(* CODESYS project doser.project

Project tree, tasks and I/O mapping:
  Device : CODESYS Control Win V3, 3S - Smart Software Solutions GmbH, order no. 305021, version 3.5.5.50
    application Application
      libraries: Standard, * (System)
      task MainTask (cyclic, interval t#20ms, priority 1) calls GateTest
      program PLC_PRG [ST]
      Global_variables/
        global variables GL_AI
        global variables GL_AO
        global variables GL_DI
        global variables GL_DO
      Units/
        function block AnalogHandler [ST]
        function block MotorDriver [ST]
        function block ProductHandler [ST]
        function block ProximitySensor [ST]
        function block GateDriver [ST]
      Tests/
        program Motor_test [LD]
        program Proximity_test [LD]
        program GateTest [LD]
*)

// Device/Application/Global_variables/GL_AI
VAR_GLOBAL
	load_cell_1_ai :INT;
	load_cell_2_ai :INT;
	
END_VAR

// Device/Application/Global_variables/GL_AO
VAR_GLOBAL
	doser_motor_freq_1_ao :INT;
	doser_motor_freq_2_ao :INT;
	mixer_motor_freq_ao :INT;
END_VAR

// Device/Application/Global_variables/GL_DI
VAR_GLOBAL
	doser_motor_overload_1 :BOOL;
	doser_motor_overload_2 :BOOL;
	mixer_motor_overload_1 :BOOL;
	gate_is_open :BOOL;
	emgc :BOOL;
	
END_VAR

// Device/Application/Global_variables/GL_DO
VAR_GLOBAL
	do_doser_moter_coil_1:BOOL;
	do_doser_moter_coil_3:BOOL;
	do_mixer_moter_coil :BOOL;
	do_gate_coil:BOOL;	
END_VAR

// Device/Application/Tests/GateTest
PROGRAM GateTest
VAR
	GateDriver_0: GateDriver;
	act: BOOL;
	egv: BOOL;
	open: BOOL;
	time_open: TIME;
	timeout: TIME;
	fault: BOOL;
	state_open: BOOL;
END_VAR

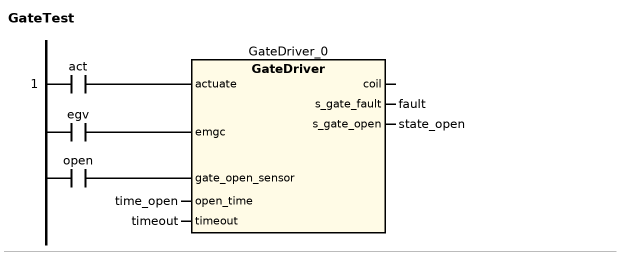
// NETWORK 1
GateDriver_0(
    actuate := act,
    emgc := egv,
    gate_open_sensor := open,
    open_time := time_open,
    timeout := timeout,
    s_gate_fault => fault,
    s_gate_open => state_open); // GateDriver

END_PROGRAM

// Device/Application/Units/GateDriver
FUNCTION_BLOCK GateDriver

VAR_INPUT
	actuate:BOOL;
	emgc:BOOL;
	gate_open_sensor:BOOL;
	open_time:TIME;
	timeout:TIME;
END_VAR


VAR_OUTPUT
	coil:BOOL;
	s_gate_fault:BOOL;
	s_gate_open:BOOL;
END_VAR


VAR
	gate_open_timeout:ton;
	gate_open_timer:ton;
	gate_trigger:r_trig;
	state:int;
END_VAR

CASE state OF
	0:
		coil:=FALSE;
		s_gate_fault:=FALSE;
		s_gate_open:=FALSE;
		gate_open_timeout(in:=FALSE);
		gate_open_timer(in:=FALSE);
		gate_trigger(clk:=actuate);
		IF gate_trigger.Q THEN
			state:=1;
			coil:=TRUE;
		END_IF
	
	1:
		gate_open_timeout(in:=TRUE, pt:=timeout);
		IF gate_open_sensor THEN
			s_gate_open:=TRUE;
			state:=2;
		ELSIF gate_open_timeout.Q THEN
			s_gate_fault:=TRUE;
			coil:=FALSE;
		END_IF
	
	2:
		gate_open_timer(in:=TRUE, pt:=open_time);
		IF gate_open_timer.Q THEN
			coil:=FALSE;
			s_gate_open:=FALSE;
		END_IF
END_CASE


IF emgc OR actuate=FALSE THEN
	state:=0;
END_IF

END_FUNCTION_BLOCK

// Device/Application/PLC_PRG
PROGRAM PLC_PRG
VAR
END_VAR

END_PROGRAM

// Device/Application/Units/AnalogHandler
FUNCTION_BLOCK AnalogHandler
VAR_INPUT
	AnalogSignal:INT;
	Gain:REAL;
	UpperLimit:REAL;
	LowerLimit:REAL;
	
END_VAR
VAR_OUTPUT
	ScaledValue:REAL;
	UpperLimitWarning:BOOL;
	LowerLimitWarning:BOOL;
END_VAR
VAR
END_VAR

ScaledValue := AnalogSignal * Gain;

IF ScaledValue > UpperLimit THEN
	UpperLimitWarning := TRUE;
ELSE
	UpperLimitWarning := FALSE;
END_IF


IF ScaledValue < LowerLimit THEN
	LowerLimitWarning := TRUE;
ELSE
	LowerLimitWarning := FALSE;
END_IF

END_FUNCTION_BLOCK

// Device/Application/Units/MotorDriver
FUNCTION_BLOCK MotorDriver

VAR_INPUT
	motor_start :BOOL;
	overload:BOOL;
	emgc:BOOL;
	feedback:BOOL;
	timeout:TIME;	
END_VAR

VAR_OUTPUT
	coil:BOOL;
	running:BOOL;
	fault:BOOL;
	timeout_warning:BOOL;	
END_VAR


VAR
	feedbackTimeout: TON;
	reset_trigger:R_TRIG;
	start: BOOL;
END_VAR

reset_trigger(clk:=start);

IF reset_trigger.q THEN
	running:=FALSE;
	fault:=FALSE;
	timeout_warning:=FALSE;
	feedbackTimeout(in:=FALSE);
END_IF


IF motor_start AND overload=FALSE AND emgc=FALSE AND timeout_warning=FALSE THEN
	coil := TRUE;
ELSE
	coil:=FALSE;
END_IF


// status
IF coil AND feedback THEN
	running:=TRUE;
ELSE
	running:=FALSE;
END_IF


IF overload OR emgc OR timeout_warning THEN
	fault:=TRUE;
ELSE
	fault:=FALSE;
END_IF


IF coil AND feedback=FALSE THEN
	feedbackTimeout(in:=TRUE, pt:=timeout);
	IF feedback=TRUE THEN
		timeout_warning:=FALSE;
		feedbackTimeout(in:=FALSE);
	ELSE
		IF feedbackTimeout.Q THEN
			timeout_warning:=TRUE;
		END_IF	
	END_IF
END_IF

END_FUNCTION_BLOCK

// Device/Application/Tests/Motor_test
PROGRAM Motor_test
VAR
	Motor:MotorDriver;
	timeout: TIME;
	running: BOOL;
	fault: BOOL;
	timeout_warning: BOOL;
	feedback: BOOL;
	overload: BOOL;
	start: BOOL;
END_VAR

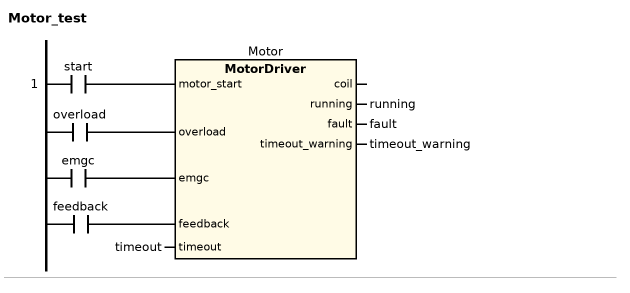
// NETWORK 1
Motor(
    motor_start := start,
    overload := overload,
    emgc := emgc,
    feedback := feedback,
    timeout := timeout,
    running => running,
    fault => fault,
    timeout_warning => timeout_warning); // MotorDriver

END_PROGRAM

// Device/Application/Units/ProductHandler
FUNCTION_BLOCK ProductHandler

VAR_INPUT
	start_dose:BOOL;
	reset:BOOL;
	current_weight:REAL;
	target_weight:REAL;
	max_weight:REAL;
	min_weight:REAL;	
END_VAR


VAR_OUTPUT
	state_done:BOOL;
	state_dosing:BOOL;
	state_max_weight_alert:BOOL;
	state_min_weight_alert:BOOL;
	state_not_enough:BOOL;
	extracted_weight:REAL;
	extra_weight:BOOL;
END_VAR


VAR
	sate:INT;
	weight:REAL;
	dose_trig:r_trig;
END_VAR

CASE state OF
	0:
		
END_CASE

END_FUNCTION_BLOCK

// Device/Application/Units/ProximitySensor
FUNCTION_BLOCK ProximitySensor

VAR_INPUT
	InputSignal :BOOL;
	on_time_delay: TIME;
	off_time_delay: TIME;		
END_VAR

VAR_OUTPUT
	detected:BOOL;	
END_VAR


VAR
	on_delay_timer:ton;
	off_delay_timer:ton;
END_VAR

on_delay_timer(in:=InputSignal, pt:=on_time_delay, q=>detected);
off_delay_timer(in:=InputSignal, pt:=off_time_delay, q=>detected);

END_FUNCTION_BLOCK

// Device/Application/Tests/Proximity_test
PROGRAM Proximity_test
VAR
	input: BOOL;
	on_time_delay: TIME;
	off_time_delay: TIME;
	sens: ProximitySensor;
END_VAR

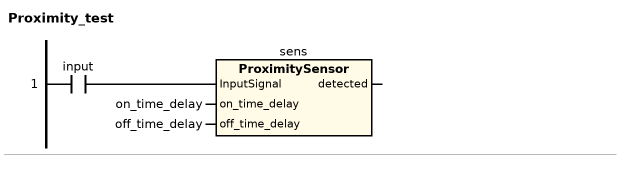
// NETWORK 1
sens(InputSignal := input, on_time_delay := on_time_delay, off_time_delay := off_time_delay); // ProximitySensor

END_PROGRAM
